FUNCTION_BLOCK FB_link
VAR_INPUT
	IN: BOOL;
END_VAR
VAR_OUTPUT
	Q: bool;
END_VAR
VAR
	fbTimerTON: TON;
	fbTimerTOF: TOF;
END_VAR

fbTimerTON(IN:= (NOT (fbTimerTOF.Q) AND IN), PT:=T#1S , Q=> fbTimerTOF.IN, ET=> );
fbTimerTOF(IN:= , PT:= fbTimerTON.PT, Q=> Q, ET=> );

END_FUNCTION_BLOCK

(* stored: Version 1.1.0.1, ProductVersion 3.1.4022.16
   POU FB_link: Id {ea086608-4b80-4aad-851a-43c59d3349dc}, SpecialFunc None *)
